RoboDK station: calibration_QKM_test.rdk

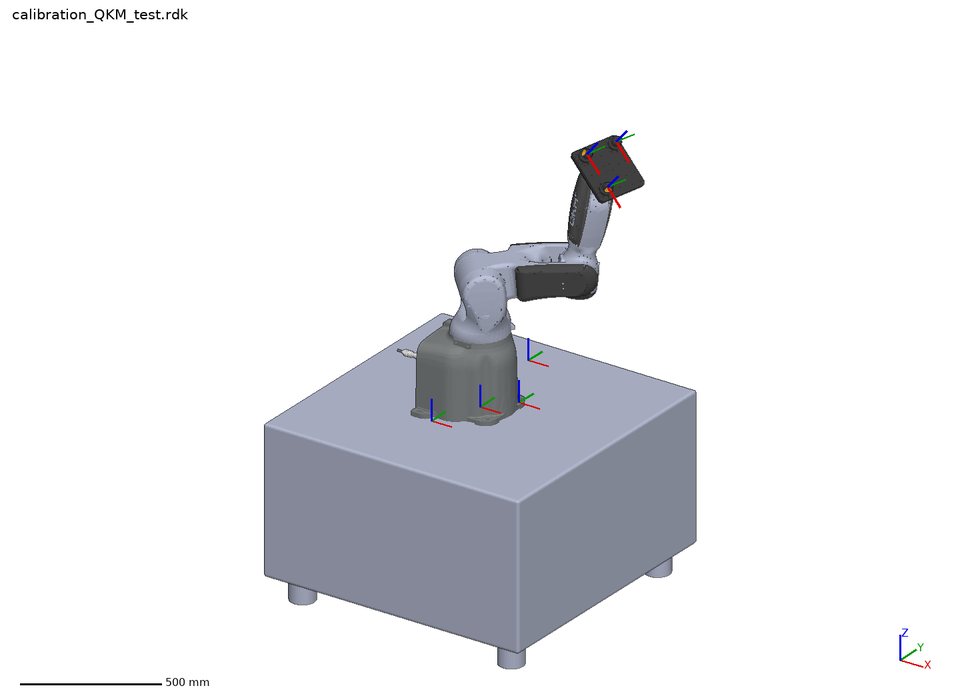
[picture v0: the station drawn from its stored meshes, robots at their saved joint values, targets as dots, program paths as lines]
Station calibration_QKM_test. Poses are relative to the parent item; angles as X-Y-Z fixed-axis rotations.
  - frame QKM HL6 Base at (0, 0, 0) mm
    - robot QKM HL6: 6 axes
        modified DH rows (alpha deg, a mm, theta deg, d mm): 0, 0, 0, 491; -90.122, 0, -89.486, 0; 0, 350, -90.184, 0; -90.964, 0, 0, 350; 89.864, 0, 0, 0; -89.694, 0, 180, 84
        joint limits [-170, -110, -136, -185, -120, -360] to [170, 110, 136, 185, 120, 360]; home [0, 0, 90, 0, 0, 0]; saved at [43.06, 85.28, -74.88, -68.67, 35.51, 16.57]
      - tool , TCP at (0, 0, 15) mm, size 210 x 210 x 65.7 mm, geometry from 2.STEP
      - frame SMR1 at (-70, -70, 42.5) mm
      - frame SMR2 at (-70, 70, 42.5) mm
      - frame SMR3 at (70, -70, 42.5) mm
    - object  at (0, 0, 0) mm, size 1100 x 1100 x 700 mm, geometry from .IGS
    - frame Base at (0, 0, 0) mm
    - frame Ref1 at (0, -297.45, 63.59) mm
    - frame Ref2 at (0, 297.05, 63.59) mm
    - frame Ref3 at (169.47, 0, 63.59) mm
  - frame Tracker Frame at (3496.69, 316.92, 766.98) mm, rotated rx 0.3 ry -1.68 rz 164.87 deg
